# B&R Automation Studio project projekt_maszyny_grawerujacej
Automation Studio 4.7.2.98; technology packages: mapp 5.10.1, mappCockpit 5.10.1, mappMotion 5.10.1, mappView 5.10.1

## Configuration Config1

CPU X20CP0484, AutomationRuntime C4.72, Build 4.1.2, Safety 0.0, Vc V4.72.0

### Task classes (Cpu.sw)
```
Cyclic#2 (cycle 20000 us, tolerance 20000 us):
  Program1 <- Program1.prg
DataObjects: McAcpSys
NcDataObjects: IProg <- CNC.IProg.dob, isProg <- CNC.isProg.dob, WProg <- CNC.WProg.dob, UProg <- CNC.UProg.dob, XProg <- CNC.XProg.dob, RProg <- CNC.RProg.dob
Binaries: arcoal, arflatprv, arsvcreg, mvLoader, TCLang, TCData, McAcpSim, FWRules, McAcpDrv, udbdef, McMechSys, mCoWebSc, Config_3, arconfig, Settings, User, asfw, ashwd, Config_6, Config_1, ashwac, TC, Role, sysconf, Config_4, Config, Hierarchy, iomap, Config_2, Config_5
Libraries: McBase, MpCnc, MpBase, McAxGroup, McPathGen, McAxis, McProgInt, McAcpAx, MpAxis, CoTrace, AsZip, FileIO, runtime, MpAlarmX, astime, MpFile, MpServer, sys_lib, asarlog, asmem, asbrstr, asieccon, aruser, dataobj, powerlnk, asusb, brsystem, asarprof, arssl
```

### Hardware
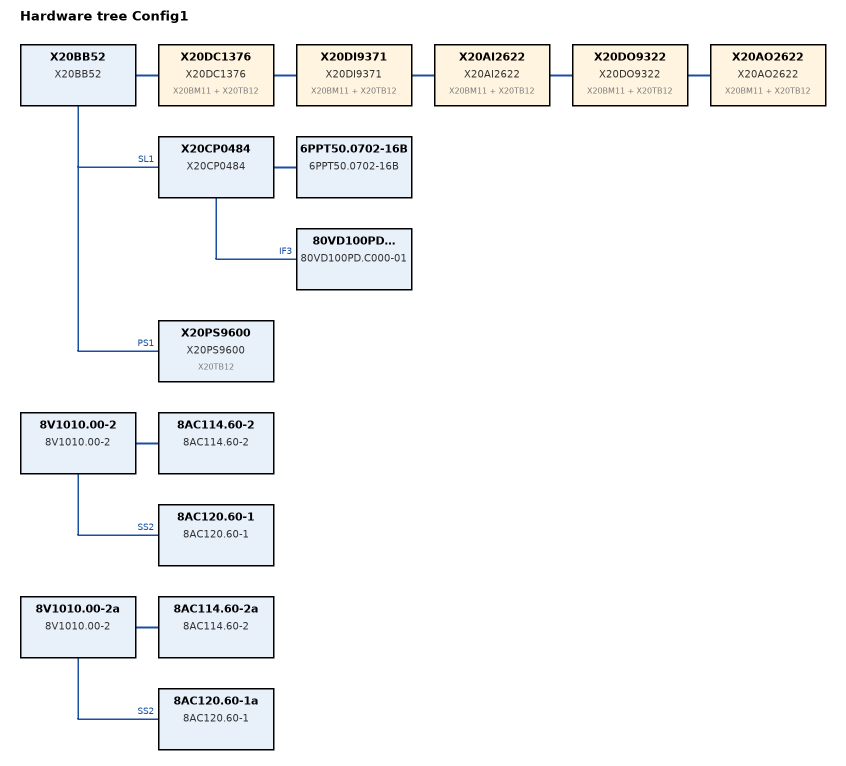
```
6PPT50.0702-16B : 6PPT50.0702-16B v1.0.0.0  [ETH1 -> X20CP0484.IF2 [Cable Type=PowerlinkCable, Length=10, Version=1.0.0.2]]
  Terminal = true
  PasswordVNC = 
  PasswordCIFS = 
  PasswordService = 
80VD100PD.C000-01 : 80VD100PD.C000-01 v2.4.0.0  [PLK1 -> X20CP0484.IF3 (NodeNumber=3) [Cable Type=PowerlinkCable, Length=10, Version=1.0.0.2]; PLK2 -> 8AC114.60-2a.PLK1 (NodeNumber=3) [Cable Type=PowerlinkCable, Length=10, Version=1.0.0.2]]
  DriveConfiguration/Module:
    McAcoposTypeID = AcoposMicroDConfig
    ActivateACOPOSSimulationOnPLC = 0
  DriveConfiguration/Channel[1]/RealAxis:
    AxisReference = gAxisQX
  DriveConfiguration/Channel[1]/RealAxis/MechanicalElements/Gearbox:
    InputIsReadOnly = 0
    Input = 1
    OutputIsReadOnly = 0
    Output = 1
  DriveConfiguration/Channel[1]/RealAxis/MechanicalElements/RotaryToLinearTransformation:
    ReferenceDistanceIsReadOnly = 0
    ReferenceDistance = 600
  DriveConfiguration/Channel[1]/RealAxis/Controller:
    ModeIsReadOnly = 0
    Mode = PositionController
  DriveConfiguration/Channel[1]/RealAxis/Controller/Mode/Position:
    ProportionalGain = 50.0
    IntegrationTime = 0.0
    PredictionTime = 0.0004
    TotalDelayTime = 0.0004
  DriveConfiguration/Channel[1]/RealAxis/Controller/Mode/Speed:
    ProportionalGainIsReadOnly = 0
    ProportionalGain = 2.0
    IntegrationTimeIsReadOnly = 0
    IntegrationTime = 0.0
    FilterTimeIsReadOnly = 0
    FilterTime = 0.0
  DriveConfiguration/Channel[1]/RealAxis/Controller/Mode/LoopFilters:
    LoopFilter1 = NotUsed
    LoopFilter2 = NotUsed
    LoopFilter3 = NotUsed
  DriveConfiguration/Channel[1]/RealAxis/Homing:
    Mode = Direct
  DriveConfiguration/Channel[1]/RealAxis/Homing/Mode:
    Position = 0.0
    ReferencePulse = NotUsed
  DriveConfiguration/Channel[1]/RealAxis/Homing:
    RestorePositionVariable = 
  DriveConfiguration/Channel[1]/RealAxis/StopReaction:
    Quickstop = DecelerationLimit
    DriveError = DecelerationLimit
  DriveConfiguration/Channel[1]/RealAxis/MovementErrorLimits:
    PositionError = 12.0
    VelocityErrorMonitoring = Automatic1
  DriveConfiguration/Channel[1]/RealAxis:
    JerkFilter = NotUsed
  DriveConfiguration/Channel[1]/RealAxis/DigitalInputs/HomingSwitch:
    Source = NotUsed
    Level = High
  DriveConfiguration/Channel[1]/RealAxis/DigitalInputs/PositiveLimitSwitch:
    Source = NotUsed
    Level = High
  DriveConfiguration/Channel[1]/RealAxis/DigitalInputs/NegativeLimitSwitch:
    Source = NotUsed
    Level = High
  DriveConfiguration/Channel[1]/RealAxis/DigitalInputs/Trigger1:
    Level = High
  DriveConfiguration/Channel[1]/RealAxis/DigitalInputs/Trigger2:
    Level = High
  DriveConfiguration/Channel[1]/RealAxis/DigitalInputs/Quickstop:
    Input = Trigger2
  DriveConfiguration/Channel[1]/RealAxis/Simulation:
    SimulationModeOnPLC = SetValueGeneration
    SimulationModeOnACOPOS = NotUsed
  DriveConfiguration/Channel[2]/RealAxis:
    AxisReference = gAxisQY
  DriveConfiguration/Channel[2]/RealAxis/MechanicalElements/Gearbox:
    InputIsReadOnly = 0
    Input = 1
    OutputIsReadOnly = 0
    Output = 1
  DriveConfiguration/Channel[2]/RealAxis/MechanicalElements/RotaryToLinearTransformation:
    ReferenceDistanceIsReadOnly = 0
    ReferenceDistance = 50
  DriveConfiguration/Channel[2]/RealAxis/Controller:
    ModeIsReadOnly = 0
    Mode = PositionController
  DriveConfiguration/Channel[2]/RealAxis/Controller/Mode/Position:
    ProportionalGain = 50.0
    IntegrationTime = 0.0
    PredictionTime = 0.0004
    TotalDelayTime = 0.0004
  DriveConfiguration/Channel[2]/RealAxis/Controller/Mode/Speed:
    ProportionalGainIsReadOnly = 0
    ProportionalGain = 2.0
    IntegrationTimeIsReadOnly = 0
    IntegrationTime = 0.0
    FilterTimeIsReadOnly = 0
    FilterTime = 0.0
  DriveConfiguration/Channel[2]/RealAxis/Controller/Mode/LoopFilters:
    LoopFilter1 = NotUsed
    LoopFilter2 = NotUsed
    LoopFilter3 = NotUsed
  DriveConfiguration/Channel[2]/RealAxis/Homing:
    Mode = Direct
  DriveConfiguration/Channel[2]/RealAxis/Homing/Mode:
    Position = 0.0
    ReferencePulse = NotUsed
  DriveConfiguration/Channel[2]/RealAxis/Homing:
    RestorePositionVariable = 
  DriveConfiguration/Channel[2]/RealAxis/StopReaction:
    Quickstop = DecelerationLimit
    DriveError = DecelerationLimit
  DriveConfiguration/Channel[2]/RealAxis/MovementErrorLimits:
    PositionError = 12.0
    VelocityErrorMonitoring = Automatic1
  DriveConfiguration/Channel[2]/RealAxis:
    JerkFilter = NotUsed
  DriveConfiguration/Channel[2]/RealAxis/DigitalInputs/HomingSwitch:
    Source = NotUsed
    Level = High
  DriveConfiguration/Channel[2]/RealAxis/DigitalInputs/PositiveLimitSwitch:
    Source = NotUsed
    Level = High
  DriveConfiguration/Channel[2]/RealAxis/DigitalInputs/NegativeLimitSwitch:
    Source = NotUsed
    Level = High
  DriveConfiguration/Channel[2]/RealAxis/DigitalInputs/Trigger1:
    Level = High
  DriveConfiguration/Channel[2]/RealAxis/DigitalInputs/Trigger2:
    Level = High
  DriveConfiguration/Channel[2]/RealAxis/DigitalInputs/Quickstop:
    Input = Trigger2
  DriveConfiguration/Channel[2]/RealAxis/Simulation:
    SimulationModeOnPLC = SetValueGeneration
    SimulationModeOnACOPOS = NotUsed
8AC114.60-2 : 8AC114.60-2 v1.0.0.8  [SS -> 8V1010.00-2.SS1; PLK1 -> 8AC114.60-2a.PLK2 [Cable Type=PowerlinkCable, Length=10, Version=1.0.0.2]]
8AC114.60-2a : 8AC114.60-2 v1.0.0.8  [SS -> 8V1010.00-2a.SS1; PLK1 -> 80VD100PD.C000-01.PLK2 [Cable Type=PowerlinkCable, Length=10, Version=1.0.0.2]; PLK2 -> 8AC114.60-2.PLK1 [Cable Type=PowerlinkCable, Length=10, Version=1.0.0.2]]
8AC120.60-1 : 8AC120.60-1 v2.2.0.0  [SS -> 8V1010.00-2.SS2]
  PlugInType = Encoder
  McAcoposTypeID = AcoposPlugInConfig
8AC120.60-1a : 8AC120.60-1 v2.2.0.0  [SS -> 8V1010.00-2a.SS2]
  PlugInType = Encoder
  McAcoposTypeID = AcoposPlugInConfig
8V1010.00-2 : 8V1010.00-2 v2.2.0.0
  DriveConfiguration/Module:
    McAcoposTypeID = AcoposConfig
    ActivateACOPOSSimulationOnPLC = 0
  DriveConfiguration/Channel[1]/RealAxis:
    AxisReference = gAxisQS
  DriveConfiguration/Channel[1]/RealAxis/MechanicalElements/Gearbox:
    InputIsReadOnly = 0
    Input = 1
    OutputIsReadOnly = 0
    Output = 1
  DriveConfiguration/Channel[1]/RealAxis/MechanicalElements/RotaryToLinearTransformation:
    ReferenceDistanceIsReadOnly = 0
    ReferenceDistance = 600
  DriveConfiguration/Channel[1]/RealAxis/Controller:
    ModeIsReadOnly = 0
    Mode = PositionController
  DriveConfiguration/Channel[1]/RealAxis/Controller/Mode/Position:
    ProportionalGain = 50.0
    IntegrationTime = 0.0
    PredictionTime = 0.0004
    TotalDelayTime = 0.0004
  DriveConfiguration/Channel[1]/RealAxis/Controller/Mode/Speed:
    ProportionalGainIsReadOnly = 0
    ProportionalGain = 2.0
    IntegrationTimeIsReadOnly = 0
    IntegrationTime = 0.0
    FilterTimeIsReadOnly = 0
    FilterTime = 0.0
  DriveConfiguration/Channel[1]/RealAxis/Controller/Mode/LoopFilters:
    LoopFilter1 = NotUsed
    LoopFilter2 = NotUsed
    LoopFilter3 = NotUsed
  DriveConfiguration/Channel[1]/RealAxis/Homing:
    Mode = Direct
  DriveConfiguration/Channel[1]/RealAxis/Homing/Mode:
    Position = 0.0
    ReferencePulse = NotUsed
  DriveConfiguration/Channel[1]/RealAxis/Homing:
    RestorePositionVariable = 
  DriveConfiguration/Channel[1]/RealAxis/StopReaction:
    Quickstop = DecelerationLimit
    DriveError = DecelerationLimit
  DriveConfiguration/Channel[1]/RealAxis/MovementErrorLimits:
    PositionError = 12.0
    VelocityErrorMonitoring = Automatic1
  DriveConfiguration/Channel[1]/RealAxis:
    JerkFilter = NotUsed
  DriveConfiguration/Channel[1]/RealAxis/DigitalInputs/HomingSwitch:
    Level = High
  DriveConfiguration/Channel[1]/RealAxis/DigitalInputs/PositiveLimitSwitch:
    Level = High
  DriveConfiguration/Channel[1]/RealAxis/DigitalInputs/NegativeLimitSwitch:
    Level = High
  DriveConfiguration/Channel[1]/RealAxis/DigitalInputs/Trigger1:
    Level = High
  DriveConfiguration/Channel[1]/RealAxis/DigitalInputs/Trigger2:
    Level = High
  DriveConfiguration/Channel[1]/RealAxis/DigitalInputs/Quickstop:
    Input = Trigger2
  DriveConfiguration/Channel[1]/RealAxis/Simulation:
    SimulationModeOnPLC = SetValueGeneration
    SimulationModeOnACOPOS = NotUsed
8V1010.00-2a : 8V1010.00-2 v2.2.0.0
  DriveConfiguration/Module:
    McAcoposTypeID = AcoposConfig
    ActivateACOPOSSimulationOnPLC = 0
  DriveConfiguration/Channel[1]/RealAxis:
    AxisReference = gAxisQZ
  DriveConfiguration/Channel[1]/RealAxis/MechanicalElements/Gearbox:
    InputIsReadOnly = 0
    Input = 1
    OutputIsReadOnly = 0
    Output = 1
  DriveConfiguration/Channel[1]/RealAxis/MechanicalElements/RotaryToLinearTransformation:
    ReferenceDistanceIsReadOnly = 0
    ReferenceDistance = 50
  DriveConfiguration/Channel[1]/RealAxis/Controller:
    ModeIsReadOnly = 0
    Mode = PositionController
  DriveConfiguration/Channel[1]/RealAxis/Controller/Mode/Position:
    ProportionalGain = 50.0
    IntegrationTime = 0.0
    PredictionTime = 0.0004
    TotalDelayTime = 0.0004
  DriveConfiguration/Channel[1]/RealAxis/Controller/Mode/Speed:
    ProportionalGainIsReadOnly = 0
    ProportionalGain = 2.0
    IntegrationTimeIsReadOnly = 0
    IntegrationTime = 0.0
    FilterTimeIsReadOnly = 0
    FilterTime = 0.0
  DriveConfiguration/Channel[1]/RealAxis/Controller/Mode/LoopFilters:
    LoopFilter1 = NotUsed
    LoopFilter2 = NotUsed
    LoopFilter3 = NotUsed
  DriveConfiguration/Channel[1]/RealAxis/Homing:
    Mode = Direct
  DriveConfiguration/Channel[1]/RealAxis/Homing/Mode:
    Position = 300.0
    ReferencePulse = NotUsed
  DriveConfiguration/Channel[1]/RealAxis/Homing:
    RestorePositionVariable = 
  DriveConfiguration/Channel[1]/RealAxis/StopReaction:
    Quickstop = DecelerationLimit
    DriveError = DecelerationLimit
  DriveConfiguration/Channel[1]/RealAxis/MovementErrorLimits:
    PositionError = 12.0
    VelocityErrorMonitoring = Automatic1
  DriveConfiguration/Channel[1]/RealAxis:
    JerkFilter = NotUsed
  DriveConfiguration/Channel[1]/RealAxis/DigitalInputs/HomingSwitch:
    Level = High
  DriveConfiguration/Channel[1]/RealAxis/DigitalInputs/PositiveLimitSwitch:
    Level = High
  DriveConfiguration/Channel[1]/RealAxis/DigitalInputs/NegativeLimitSwitch:
    Level = High
  DriveConfiguration/Channel[1]/RealAxis/DigitalInputs/Trigger1:
    Level = High
  DriveConfiguration/Channel[1]/RealAxis/DigitalInputs/Trigger2:
    Level = High
  DriveConfiguration/Channel[1]/RealAxis/DigitalInputs/Quickstop:
    Input = Trigger2
  DriveConfiguration/Channel[1]/RealAxis/Simulation:
    SimulationModeOnPLC = SetValueGeneration
    SimulationModeOnACOPOS = NotUsed
X20AI2622 : X20AI2622 v1.0.4.0  [SS1 -> X20TB12d.SS; SL -> X20BM11c.SL1]
X20AO2622 : X20AO2622 v1.1.0.0  [SS1 -> X20TB12e.SS; SL -> X20BM11d.SL1]
X20BB52 : X20BB52 v1.1.0.0
X20BM11 : X20BM11 v1.0.0.1  [X2X1 -> X20BM11b.X2X2]
X20BM11a : X20BM11 v1.0.0.1  [X2X1 -> X20BM11c.X2X2]
X20BM11b : X20BM11 v1.0.0.1  [X2X1 -> X20BB52.IF6]
X20BM11c : X20BM11 v1.0.0.1  [X2X1 -> X20BM11.X2X2]
X20BM11d : X20BM11 v1.0.0.1  [X2X1 -> X20BM11a.X2X2]
X20CP0484 : X20CP0484 v1.2.1.0  [SL -> X20BB52.SL1]
  Connector IF2:
    ActivateDevice = 1
  Connector IF3:
    InternetAddress = 10.0.0.10
  ConfigurationID = projekt_maszyny_grawerującej_Config1
  UserPartitionSize = 2
  AutomaticTransferOfUserfiles = on
  Simulation = 1
  TimerDeviceType = EPLX2X
  TimerDevice = X20CP0484.IF3
  TaskClassIdleTime = 2000
  Cyclic1Duration = 2000
  Cyclic1Tolerance = 0
  Cyclic1Stack = 32000
  Cyclic2Duration = 20000
  Cyclic2Tolerance = 20000
  Cyclic3Duration = 50000
  Cyclic3Tolerance = 50000
  Cyclic4Duration = 100000
  Cyclic4Tolerance = 100000
  Cyclic5Duration = 200000
  Cyclic5Tolerance = 200000
  Cyclic6Duration = 500000
  Cyclic6Tolerance = 500000
  Cyclic7Duration = 1000000
  Cyclic7Tolerance = 1000000
  Cyclic8Duration = 10000
  Cyclic8Tolerance = 30000000
  ActivateSntpServer = 1
  ActivateSntp = 1
  SntpcServAddr2 = 10.0.0,5
  ActivateOpcUa = 1
  OpcUaInformationModels_PV_Version = 1
X20DC1376 : X20DC1376 v1.0.2.0  [SS1 -> X20TB12c.SS; SL -> X20BM11b.SL1]
X20DI9371 : X20DI9371 v1.0.2.0  [SS1 -> X20TB12a.SS; SL -> X20BM11.SL1]
X20DO9322 : X20DO9322 v1.1.0.0  [SS1 -> X20TB12b.SS; SL -> X20BM11a.SL1]
X20PS9600 : X20PS9600 v1.0.1.0  [PS -> X20BB52.PS1; SS1 -> X20TB12.SS]
X20TB12 : X20TB12 v1.0.0.0
X20TB12a : X20TB12 v1.0.0.0
X20TB12b : X20TB12 v1.0.0.0
X20TB12c : X20TB12 v1.0.0.0
X20TB12d : X20TB12 v1.0.0.0
X20TB12e : X20TB12 v1.0.0.0
```

### IoMap.iom - X20CP0484/IoMap.iom
```iecst
VAR_CONFIG
	::gdoProcessLamp AT %QX."X20DO9322".DigitalOutput01;
	::gdoMillingLamp AT %QX."X20DO9322".DigitalOutput02;
	::Program1:Sensor AT %IX."X20DI9371".DigitalInput01;
END_VAR
```

### Config_1.axesgroup - X20CP0484/mappMotion/3AxesCNCXYZ/Config_1.axesgroup
```
Element gCncXYZ (Type=axesgroup)
  Type = PathGenAxesGroup
    ProcessingTaskClass = 1
    License = 1
    PhysicalAxes:
      JointAxes:
        JointAxis[1]:
          Name = QX
          AxisRef = gAxisQX
        JointAxis[2]:
          Name = QY
          AxisRef = gAxisQY
        JointAxis[3]:
          Name = QZ
          AxisRef = gAxisQZ
      SlaveAxes:
        SlaveAxis[1]:
          Name = QS
          AxisRef = gAxisQS
    MechanicalSystem:
      MechSysRef = MechSys_3AxCNCXYZ
    BasicSettings:
      ModalDataBehaviour = ResetToDefault
      GeometryPlanning:
        RoundingMode = Standard
        MaxCornerDeviation = 0.0
        MaxTangentialTransitionDeviation = 0.0
        MaxRadiusDeviation = 0.001
        WorkingPlane = XY
      TrajectoryPlanning = Basic
        LimitCheckResolution = UserDefinedTime
          Time = 0.01
        BufferTime = UserDefinedTime
          Time = 0.1
    AxesGroupFeatures:
      FeatureRef[1] = Feature_Programs
      FeatureRef[2] = Feature_Jogging
      FeatureRef[3] = Feature_spindles
  Alarms = None
```

### Config_2.axis - X20CP0484/mappMotion/3AxesCNCXYZ/Config_2.axis
```
Element gAxisQX (Type=axis)
  BaseTypeIsReadOnly = 0
  BaseType = Linear
    MeasurementUnit = 5066068
    MeasurementResolutionIsReadOnly = 0
    MeasurementResolution = 0.01
    CountDirectionIsReadOnly = 0
    CountDirection = Standard
  MovementLimitsIsReadOnly = 0
  MovementLimits = Internal
    Position:
      LowerLimitMin = -1.79769313486231E308
      UpperLimitMax = 1.79769313486231E308
      LowerLimit = -1000.0
      UpperLimit = 1000.0
    VelocityIsReadOnly = 0
    Velocity:
      VelocityMax = 3.4E38
      Velocity = 10000.0
    AccelerationIsReadOnly = 0
    Acceleration:
      AccelerationMax = 3.4E38
      Acceleration = 100000.0
    DecelerationIsReadOnly = 0
    Deceleration:
      DecelerationMax = 3.4E38
      Deceleration = 100000.0
  Alarms = MpAlarmX
Element gAxisQY (Type=axis)
  BaseTypeIsReadOnly = 0
  BaseType = LinearBounded
    MeasurementUnit = 5066068
    MeasurementResolutionIsReadOnly = 0
    MeasurementResolution = 0.01
    CountDirectionIsReadOnly = 0
    CountDirection = Standard
  MovementLimitsIsReadOnly = 0
  MovementLimits = Internal
    Position:
      LowerLimitMin = -1.79769313486231E308
      UpperLimitMax = 1.79769313486231E308
      LowerLimit = -100.0
      UpperLimit = 400.0
    VelocityIsReadOnly = 0
    Velocity:
      VelocityMax = 3.4E38
      Velocity = 10000.0
    AccelerationIsReadOnly = 0
    Acceleration:
      AccelerationMax = 3.4E38
      Acceleration = 100000.0
    DecelerationIsReadOnly = 0
    Deceleration:
      DecelerationMax = 3.4E38
      Deceleration = 100000.0
  Alarms = MpAlarmX
Element gAxisQZ (Type=axis)
  BaseTypeIsReadOnly = 0
  BaseType = LinearBounded
    MeasurementUnit = 5066068
    MeasurementResolutionIsReadOnly = 0
    MeasurementResolution = 0.01
    CountDirectionIsReadOnly = 0
    CountDirection = Standard
  MovementLimitsIsReadOnly = 0
  MovementLimits = Internal
    Position:
      LowerLimitMin = -1.79769313486231E308
      UpperLimitMax = 1.79769313486231E308
      LowerLimit = 0
      UpperLimit = 300
    VelocityIsReadOnly = 0
    Velocity:
      VelocityMax = 3.4E38
      Velocity = 10000.0
    AccelerationIsReadOnly = 0
    Acceleration:
      AccelerationMax = 3.4E38
      Acceleration = 100000.0
    DecelerationIsReadOnly = 0
    Deceleration:
      DecelerationMax = 3.4E38
      Deceleration = 100000.0
  Alarms = MpAlarmX
Element gAxisQS (Type=axis)
  BaseTypeIsReadOnly = 0
  BaseType = Rotary
    MeasurementUnitIsReadOnly = 0
    MeasurementUnit = 5059636
    MeasurementResolutionIsReadOnly = 0
    MeasurementResolution = 0.01
    CountDirectionIsReadOnly = 0
    CountDirection = Standard
  MovementLimitsIsReadOnly = 0
  MovementLimits = Internal
    Position:
      LowerLimitMin = -1.79769313486231E308
      UpperLimitMax = 1.79769313486231E308
      LowerLimit = -1000.0
      UpperLimit = 1000.0
    VelocityIsReadOnly = 0
    Velocity:
      VelocityMax = 3.4E38
      Velocity = 250.0
    AccelerationIsReadOnly = 0
    Acceleration:
      AccelerationMax = 3.4E38
      Acceleration = 500.0
    DecelerationIsReadOnly = 0
    Deceleration:
      DecelerationMax = 3.4E38
      Deceleration = 500.0
  Alarms = MpAlarmX
```

### Config_3.mechanicalsystem - X20CP0484/mappMotion/3AxesCNCXYZ/Config_3.mechanicalsystem
```
Element MechSys_3AxCNCXYZ (Type=mechanicalsystem)
  Type = 3AxesCNC
    Subtype = 3AxesCNCXYZ
      CoordinatesNames = Default
        XCoordinateName = X
        YCoordinateName = Y
        ZCoordinateName = Z
      WireFrameModel = Standard
        FlangeToTcp = ConnectionLine
          Distance = 0.0
      JointAxesPositionLimits:
        JointAxis[1] = UseAxisLimits
        JointAxis[2] = UseAxisLimits
        JointAxis[3] = UseAxisLimits
```

### Config_4.axesgroupfeature - X20CP0484/mappMotion/3AxesCNCXYZ/Config_4.axesgroupfeature
```
Element Feature_Programs (Type=axesgroupfeature)
  Type = Program
    ModalDataBehaviour = UseAxesGroupSettings
    InitialSettings:
      InterpolationTypes = LinearRapid
      PositionCoordinates = Absolute
      CircleCoordinates = Relative
      JACS_ACSProgramming = JACS
      ContourConnection = Inactive
      ProgrammingUnits = UseAxesGroupSettings
      Feedrates:
        FeedCharacteristic = StandardCharacteristic
        FeedType = Feedrate
        FeedReduction = Inactive
        FeedrateValue = 0.0
        InverseFeedrateValue = 0.0
        FeedratePerRevValue = 0.0
    DefaultLanguage = BRGCode
    Location = Default
      FileDevice = CNC_PrgDir
Element Feature_Jogging (Type=axesgroupfeature)
  Type = Jogging
Element Feature_spindles (Type=axesgroupfeature)
  Type = Spindles
    ModalDataBehaviour = UseAxesGroupSettings
    Spindle[1]:
      SlaveAxisName = QS
```

### Config.mpalarmxcore - X20CP0484/mappServices/Config.mpalarmxcore
```
Element gAlarmXCore (Type=mpalarmxcore)
  mapp.AlarmX.Core.Configuration:
    [0]:
      Name = EmergButton
      Message = Emergency button has been pushed
      Severity = 20
    [1]:
      Name = Elem2Small
      Message = Element is too small
      Severity = 10
    [2]:
      Name = PowerOff
      Message = Unexpected  Power Off  event
      Severity = 20
```

## Logical view

Binary libraries used (declarations not repeated): operator, runtime, astime, AsIecCon, McBase, MpCnc 5.10.1, MpBase, McAxGroup 5.10.1, McPathGen 5.10.1, McAxis, McProgInt 5.10.1, McAcpAx, MpAxis, CoTrace 5.10.0, AsZip, FileIO, MpAlarmX 5.10.1, MpFile 5.10.1, MpServer 5.10.0

### Global.typ - Global data types
```iecst
TYPE
	InType : 	STRUCT
		gdiStopButton : BOOL; (*emergency mechine stopping (INPUT)*)
		gdiObjSensor : BOOL; (*the vaule is TRUE if sensor detects object (INPUT)*)
	END_STRUCT;
	OutType : 	STRUCT
		gdoMillingLamp : BOOL; (*Lamp is on ig milling cutter is revolving (OUTPUT)*)
		gdoProcessLamp : BOOL; (*Lamp is ON if obj is being processed (OUTPUT)*)
	END_STRUCT;
END_TYPE
```

### Global.var - Global variables
```iecst
VAR
	gdiStopButton : BOOL; (*emergency mechine stopping (INPUT)*)
	gdiObjSensor : BOOL; (*the vaule is TRUE if sensor detects object (INPUT)*)
	gdoMillingLamp : BOOL; (*Lamp is on ig milling cutter is revolving (OUTPUT)*)
	gdoProcessLamp : BOOL; (*Lamp is ON if obj is being processed (OUTPUT)*)
END_VAR
```


### Program Logical/Program1 (IEC)

#### Types.typ
```iecst
TYPE
	JogStatusEnum :
		(
		JOGTYPE,
		XUP,
		XDOWN,
		YUP,
		YDOWN,
		ZUP,
		ZDOWN
		);
	WorkingModeEnum :
		(
		CHOOSE_MODE,
		AUTOMATIC,
		MANUAL,
		STOP
		);
	ServoStatusEnum :
		(
		POWER_OFF := 0,
		POWER_ON := 1,
		HOME := 2,
		READY_TO_WORK := 3
		);
	AutoModeStatusEnum :
		(
		XMOVING,
		WORKING,
		ASIGNSTART,
		CALCSIZE,
		ASIGNEND
		);
	ChooseProgrEnum :
		(
		CAPITAL_I := 0,
		SMALL_I := 1,
		CAPITAL_W := 2,
		CAPITAL_U := 3,
		CAPITAL_X := 4,
		CAPITAL_R := 5
		);
	ManualModeStatusEnum :
		(
		JOG,
		PRECISE
		);
	AsignPropEnum :
		(
		AXIS2MOVE,
		MOVEX,
		MOVEY,
		MOVEZ,
		MOVES
		);
END_TYPE
```

#### Variables.var
```iecst
(*axis and program configuration and functionality*)
VAR
	MpCnc3Axis_0 : MpCnc3Axis; (*3 axis Group*)
	Xaxis : MpAxisBasic; (*X axis func*)
	Yaxis : MpAxisBasic; (*Y axis func*)
	Zaxis : MpAxisBasic; (*Z axis func*)
	Saxis : MpAxisBasic; (*S axis func*)
	CncParameters_3Axis : MpCnc3AxisParType; (*axis group parameters*)
	X_param : MpAxisBasicParType; (*X axis parameters*)
	Y_param : MpAxisBasicParType; (*Y axis parameters*)
	Z_param : MpAxisBasicParType; (*Z axis parameters*)
	S_param : MpAxisBasicParType; (*S axis parameters*)
	ServoStatus : ServoStatusEnum; (*machine states*)
	WorkingMode : WorkingModeEnum; (*woking mode states*)
END_VAR
(*automatic mode*)
VAR
	AutoModeStatus : AutoModeStatusEnum; (*automatic mode states*)
	ChooseProgr : ChooseProgrEnum; (*enum with cnc programs*)
	StopMode : BOOL; (*ON/OFF stop mode*)
	AutomaticON : BOOL; (*ON/OFF automatic mode*)
	Sensor : BOOL; (*Sensor on off*)
	LengthStart : LREAL; (*start obj position*)
	LengthEnd : LREAL; (*end obj position*)
	ChooseElemNumber : USINT;
	Elements2Done : INT; (*processed elements*)
	NumOfElem : INT; (*Choose number of elem to process*)
	ObjLength : LREAL; (*length of obj*)
	CentreX : LREAL; (*obj centre X axis*)
END_VAR
VAR CONSTANT
	CentreY : LREAL := 200; (*obj centre Y axis*)
END_VAR
(*manual mode*)
VAR
	ManualON : BOOL; (*ON/oFF Manual mode*)
	ManualModeStatus : ManualModeStatusEnum; (*manual mode states*)
	ManXPos : LREAL; (*choose x pos*)
	ManYPos : LREAL; (*choose y pos*)
	ManZPos : LREAL; (*choose z pos*)
	ManSPos : LREAL; (*choose s pos*)
	ManXVel : REAL; (*choose x vel*)
	AsignProp : AsignPropEnum; (*states in which y can choose axis to move in manual mode*)
	ManYVel : REAL; (*choose y vel*)
	ManZVel : REAL; (*choose z vel*)
	ManSVel : REAL; (*choose s vel*)
	X2Move : BOOL; (*choose x axis to move*)
	Y2Move : BOOL; (*choose y axis to move*)
	Z2Move : BOOL; (*choose z axis to move*)
	S2Move : BOOL; (*choose s axis to move*)
	Moveaxis : BOOL; (*comfirms axis move in manual mode*)
END_VAR
(*jogging*)
VAR
	JogStatus : JogStatusEnum; (*jog mode states*)
	JogUpX : BOOL; (*jog x forward*)
	JogDownX : BOOL; (*jog x backward*)
	JogUpY : BOOL; (*jog y forward*)
	JogDownY : BOOL; (*jog y backward*)
	JogUpZ : BOOL; (*jog z gorward*)
	JogDownZ : BOOL; (*jog z backward*)
	JogUpS : BOOL; (*jog s forward*)
	JogDownS : BOOL; (*jog s backward*)
	JogModeOn : BOOL; (*on offf joging mode*)
END_VAR
(*visualization (variables needed to show process icons)*)
VAR
	Proccessing : BOOL;
	YOff : BOOL;
	Ymove : BOOL;
	YOn : BOOL;
	XOff : BOOL;
	Xmove : BOOL;
	XOn : BOOL;
	ZOff : BOOL;
	Zmove : BOOL;
	ZOn : BOOL;
	SOff : BOOL;
	Smove : BOOL;
	SOn : BOOL;
	ActMode4MV : STRING[80]; (*Helps display actual mode in mappView *)
END_VAR
(*AlarmSystem*)
VAR
	EmergStop : BOOL; (*Emergency Stop Button. Stops machine *)
	MpAlarmXCore_0 : MpAlarmXCore;
END_VAR
VAR CONSTANT
	cmdErrorReset : BOOL := FALSE;
END_VAR
VAR
	SetAlarmEmerg : USINT;
	cmdSetAlarm : BOOL;
	AckALL : MpAlarmXAcknowledgeAll;
	EmergStopAck : BOOL;
	AckAllButton : BOOL;
	Elem2SmallAck : BOOL;
	Elem2Small : BOOL;
	WarningSymbol1 : BOOL;
	WarningSymbol2 : BOOL;
	ShowWarning : BOOL;
END_VAR
(*Alarm History*)
VAR
	MpAlarmXHistory_0 : MpAlarmXHistory;
	MpAlarmXHistoryUI_0 : MpAlarmXHistoryUI;
	MpAlarmXListUI_0 : MpAlarmXListUI;
	MpAlarmXListUIConnectType_0 : MpAlarmXListUIConnectType;
	AlarmXHistoryUIConnect : MpAlarmXHistoryUIConnectType;
END_VAR
(*Visualization plc Open state*)
VAR
	XState : STRING[80];
	YState : STRING[80];
	ZState : STRING[80];
	SState : STRING[80];
END_VAR
```

#### Main.st
```iecst
(*************************************************************
* COPYRIGHT – B&R Industrial Automation
 *************************************************************
* PROGRAM: Milling Machine
* Author: Patrtyk Tomaszewski
* Created: 10/8/2020
*************************************************************
* Project Milling Machine
*************************************************************)

PROGRAM _INIT
	//Alarms
	MpAlarmXCore_0.MpLink := ADR(gAlarmXCore);
	MpAlarmXCore_0.Enable := TRUE;
	AckALL.MpLink := ADR(gAlarmXCore);
	AckALL.Enable := TRUE;
	//Alarm History

	MpAlarmXHistory_0.MpLink := ADR(gAlarmXHistory);
	MpAlarmXHistory_0.Enable := TRUE;
	MpAlarmXHistory_0.DeviceName := ADR('CF');

	//3 axis
	MpCnc3Axis_0.MpLink := ADR(gCncXYZ);
	MpCnc3Axis_0.Enable := TRUE;
	MpCnc3Axis_0.Parameters := ADR(CncParameters_3Axis);
	MpCnc3Axis_0.Override := 100.0;
	///////////////////////////////

	//X axis
	Xaxis.MpLink := ADR(gAxisQX);
	Xaxis.Parameters := ADR(X_param);
	Xaxis.Enable := TRUE;
	X_param.Velocity := 30.0;
	X_param.Acceleration := 50.0;
	X_param.Deceleration := 50.0;
	X_param.Homing.Mode := mcHOMING_DEFAULT;
   /////

	//Y axis
	Yaxis.MpLink := ADR(gAxisQY);
	Yaxis.Parameters := ADR(Y_param);
	Yaxis.Enable := TRUE;
	Y_param.Velocity := 30.0;
	Y_param.Acceleration := 50.0;
	Y_param.Deceleration := 50.0;
	Y_param.Homing.Mode := mcHOMING_DEFAULT;
	/////

	//Z axis
	Zaxis.MpLink := ADR(gAxisQZ);
	Zaxis.Parameters := ADR(Z_param);
	Zaxis.Enable := TRUE;
	Z_param.Velocity := 30.0;
	Z_param.Acceleration := 50.0;
	Z_param.Deceleration := 50.0;
	Z_param.Homing.Mode := mcHOMING_DEFAULT;
	/////

	//S axis
	Saxis.MpLink := ADR(gAxisQS);
	Saxis.Parameters := ADR(S_param);
	Saxis.Enable := TRUE;
	S_param.Velocity := 166.6;
	S_param.Acceleration := 400.0;
	S_param.Deceleration := 400.0;
	S_param.Homing.Mode := mcHOMING_DEFAULT;
	S_param.Jog.Velocity := 166.6;
	S_param.Jog.Acceleration := 400.0;
	S_param.Jog.Deceleration := 400.0;

	/////

END_PROGRAM

PROGRAM _CYCLIC

	(*
	Powering On Servo*)

	CASE ServoStatus OF

		POWER_OFF:
			ActMode4MV := 'POWER OFF';
			MpCnc3Axis_0.Update := TRUE;
			Xaxis.Power := FALSE;
			Yaxis.Power := FALSE;
			Zaxis.Power := FALSE;
			Saxis.Power := FALSE;
			StopMode := FALSE;
			ManualON := FALSE;
			AutomaticON := FALSE;
			IF  MpCnc3Axis_0.Info.ReadyToPowerOn AND MpCnc3Axis_0.Power THEN
				MpCnc3Axis_0.Update := FALSE;
				ServoStatus := POWER_ON;

			END_IF

		POWER_ON:
			ActMode4MV := 'POWER ON';
			MpCnc3Axis_0.Update := TRUE;
			Xaxis.Power := TRUE;
			Yaxis.Power := TRUE;
			Zaxis.Power := TRUE;
			Saxis.Power := TRUE;
			IF  MpCnc3Axis_0.PowerOn AND Xaxis.PowerOn AND Yaxis.PowerOn AND Zaxis.PowerOn AND Saxis.PowerOn THEN;
				MpCnc3Axis_0.Update := FALSE;
				ServoStatus := HOME;

			END_IF

		HOME:
			ActMode4MV := 'Homing';
			MpCnc3Axis_0.Home := TRUE;
			IF  MpCnc3Axis_0.IsHomed AND Xaxis.Position = 0.0 AND Yaxis.Position = 0.0 AND Zaxis.Position = 300.0 THEN;
				ActMode4MV := 'Ready To Work';
				ServoStatus := READY_TO_WORK;

			END_IF
		READY_TO_WORK:
			MpCnc3Axis_0.Home := FALSE;

			CASE WorkingMode OF

				CHOOSE_MODE:
					IF AutomaticON THEN;
						WorkingMode := AUTOMATIC;
						Elements2Done := 0;
					ELSIF ManualON THEN;
						WorkingMode := MANUAL;
					END_IF

				AUTOMATIC:
					AutomaticON := TRUE;
					MpCnc3Axis_0.Power := TRUE;
					ManualON := FALSE;

					ActMode4MV := 'Automatic Mode';
					CASE AutoModeStatus OF
						////////Const X axis move until we find elem
						XMOVING:
							Elem2Small := FALSE;
							X_param.Velocity := 30.0;
							Xaxis.Update := TRUE;
							IF Sensor = FALSE THEN;
								Xaxis.Update := FALSE;
								Xaxis.MoveVelocity := TRUE;
								IF StopMode THEN
									Xaxis.MoveVelocity := FALSE;
									AutomaticON := FALSE;
									NumOfElem := 0;
									WorkingMode := STOP;

								END_IF;

							ELSE
								gdoProcessLamp := TRUE;
								AutoModeStatus := ASIGNSTART;
							END_IF
							///////////////////////////

							///Calculate Length of element

						ASIGNSTART:
							X_param.Velocity := 20.0;
							Xaxis.Update := TRUE;
							LengthStart := Xaxis.Position;
							AutoModeStatus := ASIGNEND;

						ASIGNEND:
							Xaxis.Update := FALSE;
							IF Sensor = FALSE THEN;
								LengthEnd := Xaxis.Position;
								AutoModeStatus := CALCSIZE;
							END_IF

						CALCSIZE:
							ObjLength := LengthEnd - LengthStart;
							CentreX := LengthStart + (ObjLength / 2);
							AutoModeStatus := WORKING;
							/////////////////////////////////////

							///start program
						WORKING:
							Xaxis.MoveVelocity := FALSE;
							X_param.Velocity := 30.0;
							//Program I
							IF ChooseProgr = CAPITAL_I THEN

								IF ObjLength < 40 THEN
									Elem2Small := TRUE;
									gdoProcessLamp := FALSE;
									AutoModeStatus := XMOVING;

								ELSE
									X_param.Position := CentreX;
									Xaxis.Update := TRUE;
									Xaxis.MoveAbsolute := TRUE;

									IF  Xaxis.InPosition  THEN;
										Xaxis.Update := FALSE;
										Xaxis.MoveAbsolute := FALSE;
										CncParameters_3Axis.ProgramName := 'IProg';
										MpCnc3Axis_0.Update := TRUE;
										MpCnc3Axis_0.MoveProgram := TRUE;
										IF MpCnc3Axis_0.MoveDone THEN
											MpCnc3Axis_0.Update := FALSE;
											MpCnc3Axis_0.MoveProgram := FALSE;
											X_param.Position := LengthEnd;
											Xaxis.Update := TRUE;
											Xaxis.MoveAbsolute := TRUE;
											IF Xaxis.InPosition THEN
												Xaxis.Update := FALSE;
												Xaxis.MoveAbsolute := FALSE;
												IF StopMode THEN
													AutomaticON := FALSE;
													gdoProcessLamp := FALSE;
													NumOfElem := 0;
													WorkingMode := STOP;////////going to stop mode after completing program

												ELSE
													gdoProcessLamp := FALSE;
													Elements2Done := Elements2Done + 1;
													IF (Elements2Done = NumOfElem) AND (NumOfElem <> 0.0) THEN;
														NumOfElem := 0;
														Elements2Done := 0;
														StopMode := TRUE;
														AutomaticON := FALSE;
														WorkingMode := STOP;
													ELSE
														IF NumOfElem = 0.0 THEN;
															Elements2Done := FALSE;
															AutoModeStatus := XMOVING;
														ELSE
															AutoModeStatus := XMOVING;
														END_IF;
													END_IF;
												END_IF;

											END_IF;
										END_IF;
									END_IF;
								END_IF;
								//Program i
							ELSIF ChooseProgr = SMALL_I THEN

								IF ObjLength < 40 THEN
									Elem2Small := TRUE;
									gdoProcessLamp := FALSE;
									AutoModeStatus := XMOVING;
								ELSE

									X_param.Position := CentreX;
									Xaxis.Update := TRUE;
									Xaxis.MoveAbsolute := TRUE;
									IF Xaxis.InPosition THEN;
										Xaxis.Update := FALSE;
										Xaxis.MoveAbsolute := FALSE;
										CncParameters_3Axis.ProgramName := 'isProg';
										MpCnc3Axis_0.Update := TRUE;
										MpCnc3Axis_0.MoveProgram := TRUE;
										IF MpCnc3Axis_0.MoveDone THEN
											MpCnc3Axis_0.Update := FALSE;
											MpCnc3Axis_0.MoveProgram := FALSE;
											X_param.Position := LengthEnd;
											Xaxis.Update := TRUE;
											Xaxis.MoveAbsolute := TRUE;
											IF Xaxis.InPosition THEN
												Xaxis.Update := FALSE;
												Xaxis.MoveAbsolute := FALSE;
												IF StopMode THEN
													gdoProcessLamp := FALSE;
													AutomaticON := FALSE;
													NumOfElem := 0;
													WorkingMode := STOP;////////going to stop mode after completing program
												ELSE
													gdoProcessLamp := FALSE;
													Elements2Done := Elements2Done + 1;
													IF (Elements2Done = NumOfElem) AND (NumOfElem <> 0.0) THEN;
														NumOfElem := 0;
														Elements2Done := 0;
														StopMode := TRUE;
														AutomaticON := FALSE;
														WorkingMode := STOP;
													ELSE
														IF NumOfElem = 0.0 THEN;
															Elements2Done := FALSE;
															AutoModeStatus := XMOVING;
														ELSE
															AutoModeStatus := XMOVING;
														END_IF;
													END_IF;
												END_IF;

											END_IF;
										END_IF;
									END_IF;
								END_IF;
								///Program W
							ELSIF ChooseProgr = CAPITAL_W THEN
								IF ObjLength < 140 THEN
									Elem2Small := TRUE;
									gdoProcessLamp := FALSE;
									AutoModeStatus := XMOVING;
								ELSE

									X_param.Position := CentreX + 50;
									Xaxis.Update := TRUE;
									Xaxis.MoveAbsolute := TRUE;
									IF Xaxis.InPosition THEN;
										Xaxis.Update := FALSE;
										Xaxis.MoveAbsolute := FALSE;
										CncParameters_3Axis.ProgramName := 'WProg';
										MpCnc3Axis_0.Update := TRUE;
										MpCnc3Axis_0.MoveProgram := TRUE;
										IF MpCnc3Axis_0.MoveDone THEN
											MpCnc3Axis_0.Update := FALSE;
											MpCnc3Axis_0.MoveProgram := FALSE;
											X_param.Position := LengthEnd;
											Xaxis.Update := TRUE;
											Xaxis.MoveAbsolute := TRUE;
											IF Xaxis.InPosition  THEN
												Xaxis.Update := FALSE;
												Xaxis.MoveAbsolute := FALSE;
												IF StopMode THEN
													AutomaticON := FALSE;
													gdoProcessLamp := FALSE;
													NumOfElem := 0;
													WorkingMode := STOP;////////going to stop mode after completing program
												ELSE
													gdoProcessLamp := FALSE;
													Elements2Done := Elements2Done + 1;
													IF (Elements2Done = NumOfElem) AND (NumOfElem <> 0.0) THEN;
														NumOfElem := 0;
														Elements2Done := 0;
														StopMode := TRUE;
														AutomaticON := FALSE;
														WorkingMode := STOP;
													ELSE
														IF NumOfElem = 0.0 THEN;
															Elements2Done := FALSE;
															AutoModeStatus := XMOVING;
														ELSE
															AutoModeStatus := XMOVING;
														END_IF;
													END_IF;
												END_IF;

											END_IF;
										END_IF;
									END_IF;
								END_IF;
								///Program U
							ELSIF ChooseProgr = CAPITAL_U  THEN
								IF ObjLength < 115 THEN
									Elem2Small := TRUE;
									gdoProcessLamp := FALSE;
									AutoModeStatus := XMOVING;
								ELSE

									X_param.Position := CentreX + 37.5;
									Xaxis.Update := TRUE;
									Xaxis.MoveAbsolute := TRUE;
									IF Xaxis.InPosition THEN;
										Xaxis.Update := FALSE;
										Xaxis.MoveAbsolute := FALSE;
										CncParameters_3Axis.ProgramName := 'UProg';
										MpCnc3Axis_0.Update := TRUE;
										MpCnc3Axis_0.MoveProgram := TRUE;
										IF MpCnc3Axis_0.MoveDone THEN
											MpCnc3Axis_0.Update := FALSE;
											MpCnc3Axis_0.MoveProgram := FALSE;
											X_param.Position := LengthEnd;
											Xaxis.Update := TRUE;
											Xaxis.MoveAbsolute := TRUE;
											IF Xaxis.InPosition THEN
												Xaxis.Update := FALSE;
												Xaxis.MoveAbsolute := FALSE;
												IF StopMode THEN
													AutomaticON := FALSE;
													gdoProcessLamp := FALSE;
													NumOfElem := 0;
													WorkingMode := STOP;////////going to stop mode after completing program
												ELSE
													gdoProcessLamp := FALSE;
													Elements2Done := Elements2Done + 1;
													IF (Elements2Done = NumOfElem) AND (NumOfElem <> 0.0) THEN;
														NumOfElem := 0;
														Elements2Done := 0;
														StopMode := TRUE;
														AutomaticON := FALSE;
														WorkingMode := STOP;
													ELSE
														IF NumOfElem = 0.0 THEN;
															Elements2Done := FALSE;
															AutoModeStatus := XMOVING;
														ELSE
															AutoModeStatus := XMOVING;
														END_IF;
													END_IF;
												END_IF;

											END_IF;
										END_IF;
									END_IF;
								END_IF;
								//Program X
							ELSIF ChooseProgr = CAPITAL_X THEN
								IF ObjLength < 115 THEN
									Elem2Small := TRUE;
									gdoProcessLamp := FALSE;
									AutoModeStatus := XMOVING;
								ELSE

									X_param.Position := CentreX + 37.5;
									Xaxis.Update := TRUE;
									Xaxis.MoveAbsolute := TRUE;
									IF  Xaxis.InPosition THEN;
										Xaxis.Update := FALSE;
										Xaxis.MoveAbsolute := FALSE;
										CncParameters_3Axis.ProgramName := 'XProg';
										MpCnc3Axis_0.Update := TRUE;
										MpCnc3Axis_0.MoveProgram := TRUE;
										IF MpCnc3Axis_0.MoveDone THEN;
											MpCnc3Axis_0.Update := FALSE;
											MpCnc3Axis_0.MoveProgram := FALSE;
											X_param.Position := LengthEnd;
											Xaxis.Update := TRUE;
											Xaxis.MoveAbsolute := TRUE;
											IF Xaxis.InPosition THEN
												Xaxis.Update := FALSE;
												Xaxis.MoveAbsolute := FALSE;
												IF StopMode THEN
													AutomaticON := FALSE;
													gdoProcessLamp := FALSE;
													NumOfElem := 0;
													WorkingMode := STOP;////////going to stop mode after completing program
												ELSE
													gdoProcessLamp := FALSE;
													Elements2Done := Elements2Done + 1;
													IF (Elements2Done = NumOfElem) AND (NumOfElem <> 0.0) THEN;
														NumOfElem := 0;
														Elements2Done := 0;
														StopMode := TRUE;
														AutomaticON := FALSE;
														WorkingMode := STOP;
													ELSE
														IF NumOfElem = 0.0 THEN;
															Elements2Done := FALSE;
															AutoModeStatus := XMOVING;
														ELSE
															AutoModeStatus := XMOVING;
														END_IF;
													END_IF;
												END_IF;

											END_IF;
										END_IF;
									END_IF;
								END_IF;
								//Program R
							ELSIF ChooseProgr = CAPITAL_R THEN
								IF ObjLength < 90 THEN
									Elem2Small := TRUE;
									gdoProcessLamp := FALSE;
									AutoModeStatus := XMOVING;
								ELSE

									X_param.Position := CentreX + 25;
									Xaxis.Update := TRUE;
									Xaxis.MoveAbsolute := TRUE;
									IF Xaxis.InPosition THEN;
										Xaxis.Update := FALSE;
										Xaxis.MoveAbsolute := FALSE;
										CncParameters_3Axis.ProgramName := 'RProg';
										MpCnc3Axis_0.Update := TRUE;
										MpCnc3Axis_0.MoveProgram := TRUE;
										IF MpCnc3Axis_0.MoveDone THEN
											MpCnc3Axis_0.Update := FALSE;
											MpCnc3Axis_0.MoveProgram := FALSE;
											X_param.Position := LengthEnd;
											Xaxis.Update := TRUE;
											Xaxis.MoveAbsolute := TRUE;
											IF Xaxis.InPosition  THEN;
												Xaxis.Update := FALSE;
												Xaxis.MoveAbsolute := FALSE;
												IF StopMode THEN
													AutomaticON := FALSE;
													gdoProcessLamp := FALSE;
													NumOfElem := 0;
													WorkingMode := STOP;////////going to stop mode after completing program
												ELSE
													gdoProcessLamp := FALSE;
													Elements2Done := Elements2Done + 1;
													IF (Elements2Done = NumOfElem) AND (NumOfElem <> 0.0) THEN;
														NumOfElem := 0;
														Elements2Done := 0;
														StopMode := TRUE;
														AutomaticON := FALSE;
														WorkingMode := STOP;
													ELSE
														IF NumOfElem = 0.0 THEN;
															Elements2Done := FALSE;
															AutoModeStatus := XMOVING;
														ELSE
															AutoModeStatus := XMOVING;
														END_IF;
													END_IF;
												END_IF;

											END_IF;

										END_IF;
									END_IF;
								END_IF;
							END_IF;

					END_CASE

				MANUAL:
					ManualON := TRUE;
					MpCnc3Axis_0.Power := TRUE;
					IF AutomaticON THEN;
						ManualON := FALSE;
						WorkingMode := AUTOMATIC;
						JogUpX := FALSE;
						JogDownX := FALSE;
						JogUpY := FALSE;
						JogDownY := FALSE;
						JogUpZ := FALSE;
						JogUpS := FALSE;
						Saxis.JogPositive := FALSE;
					END_IF;

					IF StopMode THEN;
						ManualON := FALSE;
						WorkingMode := STOP;
						JogUpX := FALSE;
						JogDownX := FALSE;
						JogUpY := FALSE;
						JogDownY := FALSE;
						JogUpZ := FALSE;
						JogUpS := FALSE;
						Saxis.JogPositive := FALSE;

					END_IF;

					ActMode4MV := 'Manual Mode';
					IF JogModeOn THEN;
						ManualModeStatus := JOG;
					ELSE
						ManualModeStatus := PRECISE;
					END_IF;

					CASE ManualModeStatus OF
						////Chossing which axis we want to move
						PRECISE:
							IF X2Move = FALSE AND Y2Move = FALSE AND Z2Move = FALSE AND S2Move = FALSE THEN;
								Moveaxis := FALSE;
							END_IF;
							CASE AsignProp OF
								AXIS2MOVE:
									IF X2Move THEN;
											X2Move := FALSE;
											Y2Move := FALSE;
											Z2Move := FALSE;
											S2Move := FALSE;
										AsignProp := MOVEX;
									ELSIF Y2Move THEN;
											X2Move := FALSE;
											Y2Move := FALSE;
											Z2Move := FALSE;
											S2Move := FALSE;
										AsignProp := MOVEY;
									ELSIF Z2Move THEN;
											X2Move := FALSE;
											Y2Move := FALSE;
											Z2Move := FALSE;
											S2Move := FALSE;
										AsignProp := MOVEZ;
									ELSIF S2Move THEN;
											X2Move := FALSE;
											Y2Move := FALSE;
											Z2Move := FALSE;
											S2Move := FALSE;
										AsignProp := MOVES;
									END_IF;
								MOVEX:
									IF Moveaxis THEN;

										X_param.Velocity := ManXVel;
										X_param.Position := ManXPos;
										Xaxis.MoveAbsolute := TRUE;
										Moveaxis := TRUE;
										X2Move := TRUE;
										IF Xaxis.Position = ManXPos THEN;
											Moveaxis := FALSE;
											Xaxis.MoveAbsolute := FALSE;
											X2Move := FALSE;
											AsignProp := AXIS2MOVE;
										END_IF;
									END_IF;
								MOVEY:
									IF Moveaxis THEN;
										Y2Move := TRUE;
										Y_param.Velocity := ManYVel;
										Y_param.Position := ManYPos;
										Yaxis.MoveAbsolute := TRUE;
										Moveaxis := TRUE;
										IF Yaxis.Position = ManYPos THEN;
											Moveaxis := FALSE;
											Yaxis.MoveAbsolute := FALSE;
											Y2Move := FALSE;
											AsignProp := AXIS2MOVE;
										END_IF;
									END_IF;
								MOVEZ:
									IF Moveaxis THEN;
										Z2Move := TRUE;
										Z_param.Velocity := ManZVel;
										Z_param.Position := ManZPos;
										Zaxis.MoveAbsolute := TRUE;
										Moveaxis := TRUE;
										IF Zaxis.Position = ManZPos THEN;
											Moveaxis := FALSE;
											Zaxis.MoveAbsolute := FALSE;
											Z2Move := FALSE;
											AsignProp := AXIS2MOVE;
										END_IF;
									END_IF;
								MOVES:
									IF Moveaxis THEN;
										S2Move := TRUE;
										S_param.Velocity := ManSVel;
										S_param.Position := ManSPos;
										Saxis.MoveAbsolute := TRUE;
										Moveaxis := TRUE;
										IF Saxis.Position = ManSPos THEN;
											Moveaxis := FALSE;
											Saxis.MoveAbsolute := FALSE;
											S2Move := FALSE;
											AsignProp := AXIS2MOVE;
										END_IF;
									END_IF;
							END_CASE
						JOG:
							CASE JogStatus OF
								JOGTYPE:
									IF JogUpX THEN;
										JogStatus := XUP;
									ELSIF JogDownX THEN;
										JogStatus := XDOWN;
									ELSIF JogUpY THEN;
										JogStatus := YUP;
									ELSIF JogDownY THEN;
										JogStatus := YDOWN;
									ELSIF JogUpZ THEN;
										JogStatus := ZUP;
									ELSIF JogDownZ THEN;
										JogStatus := ZDOWN;
									END_IF;
								XUP:
									JogDownX := FALSE;
									JogUpY := FALSE;
									JogDownY := FALSE;
									JogUpZ := FALSE;
									JogDownZ := FALSE;
									Xaxis.JogPositive := TRUE;
									Xaxis.JogNegative := FALSE;
									Yaxis.JogPositive := FALSE;
									Yaxis.JogNegative := FALSE;
									Zaxis.JogPositive := FALSE;
									Zaxis.JogNegative := FALSE;
									IF JogUpX = FALSE THEN;
										Xaxis.JogPositive := FALSE;
										JogStatus := JOGTYPE;
									END_IF;
								XDOWN:
									JogUpX := FALSE;
									JogUpY := FALSE;
									JogDownY := FALSE;
									JogUpZ := FALSE;
									JogDownZ := FALSE;
									Xaxis.JogPositive := FALSE;
									Xaxis.JogNegative := TRUE;
									Yaxis.JogPositive := FALSE;
									Yaxis.JogNegative := FALSE;
									Zaxis.JogPositive := FALSE;
									Zaxis.JogNegative := FALSE;
									IF JogDownX = FALSE THEN;
										Xaxis.JogNegative := FALSE;
										JogStatus := JOGTYPE;
									END_IF;
								YUP:
									JogUpX := FALSE;
									JogDownX := FALSE;
									JogDownY := FALSE;
									JogUpZ := FALSE;
									JogDownZ := FALSE;
									Xaxis.JogPositive := FALSE;
									Xaxis.JogNegative := FALSE;
									Yaxis.JogPositive := TRUE;
									Yaxis.JogNegative := FALSE;
									Zaxis.JogPositive := FALSE;
									Zaxis.JogNegative := FALSE;
									IF JogUpY = FALSE THEN;
										Yaxis.JogPositive := FALSE;
										JogStatus := JOGTYPE;
									END_IF;
								YDOWN:
									JogUpX := FALSE;
									JogDownX := FALSE;
									JogUpY := FALSE;
									JogUpZ := FALSE;
									JogDownZ := FALSE;
									Xaxis.JogPositive := FALSE;
									Xaxis.JogNegative := FALSE;
									Yaxis.JogPositive := FALSE;
									Yaxis.JogNegative := TRUE;
									Zaxis.JogPositive := FALSE;
									Zaxis.JogNegative := FALSE;
									IF JogDownY = FALSE OR (Yaxis.Position = -100.0) THEN;
										Yaxis.JogNegative := FALSE;
										JogStatus := JOGTYPE;
									END_IF;
								ZUP:
									JogUpX := FALSE;
									JogDownX := FALSE;
									JogUpY := FALSE;
									JogDownY := FALSE;
									JogDownZ := FALSE;
									Xaxis.JogPositive := FALSE;
									Xaxis.JogNegative := FALSE;
									Yaxis.JogPositive := FALSE;
									Yaxis.JogNegative := FALSE;
									Zaxis.JogPositive := TRUE;
									Zaxis.JogNegative := FALSE;
									IF JogUpZ = FALSE THEN;
										Zaxis.JogPositive := FALSE;
										JogStatus := JOGTYPE;
									END_IF;
								ZDOWN:
									JogUpX := FALSE;
									JogDownX := FALSE;
									JogUpY := FALSE;
									JogDownY := FALSE;
									JogUpZ := FALSE;
									Xaxis.JogPositive := FALSE;
									Xaxis.JogNegative := FALSE;
									Yaxis.JogPositive := FALSE;
									Yaxis.JogNegative := FALSE;
									Zaxis.JogPositive := FALSE;
									Zaxis.JogNegative := TRUE;
									IF JogDownZ = FALSE THEN;
										Zaxis.JogNegative := FALSE;
										JogStatus := JOGTYPE;
									END_IF;
							END_CASE

							IF JogUpS THEN;
								Saxis.JogPositive := TRUE;
							ELSE
								Saxis.JogPositive := FALSE;
							END_IF;

					END_CASE
					///////////
					///////////////////

					//////////////////////
					////////////////////
				STOP:
					ActMode4MV := 'STOP Mode';
					Xaxis.Stop := TRUE;
					Yaxis.Stop := TRUE;
					Zaxis.Stop := TRUE;
					Saxis.Stop := TRUE;
					IF (StopMode = FALSE) AND (Xaxis.Stop = TRUE) AND (Yaxis.Stop = TRUE) AND (Zaxis.Stop = TRUE) AND (Saxis.Stop = TRUE) THEN
						IF (AutomaticON = TRUE) AND (ManualON = FALSE) THEN;
							Xaxis.Stop := FALSE;
							Yaxis.Stop := FALSE;
							Zaxis.Stop := FALSE;
							Saxis.Stop := FALSE;
							IF (Xaxis.Stop = FALSE) AND (Yaxis.Stop = FALSE) AND (Zaxis.Stop = FALSE) AND (Saxis.Stop = FALSE) THEN;
								WorkingMode := AUTOMATIC;
								AutoModeStatus := XMOVING;
							END_IF;
						ELSIF (AutomaticON = FALSE) AND (ManualON = TRUE) THEN;
							WorkingMode := MANUAL;
							Xaxis.Stop := FALSE;
							Yaxis.Stop := FALSE;
							Zaxis.Stop := FALSE;
							Saxis.Stop := FALSE;
							IF (Xaxis.Stop = FALSE) AND (Yaxis.Stop = FALSE) AND (Zaxis.Stop = FALSE) AND (Saxis.Stop = FALSE) THEN;
								WorkingMode := MANUAL;
							END_IF;
						END_IF;
					ELSIF StopMode THEN;
						AutomaticON := FALSE;
						ManualON := FALSE;

					END_IF;
					IF EDGENEG(MpCnc3Axis_0.Power) THEN;
						AutomaticON := FALSE;
						ManualON := FALSE;
						StopMode := FALSE;
						Xaxis.Update := FALSE;
						IF MpCnc3Axis_0.PowerOn = FALSE THEN;
							WorkingMode := CHOOSE_MODE;
							ServoStatus := POWER_OFF;
							Xaxis.MoveVelocity := FALSE;
						END_IF;
					END_IF;

			END_CASE

	END_CASE;
//Emergency Button
	IF EDGEPOS (EmergStop) THEN;
		MpCnc3Axis_0.Power := FALSE;
		AutomaticON := FALSE;
		ManualON := FALSE;
		StopMode := FALSE;
		Xaxis.Update := FALSE;

	END_IF
	IF  WarningSymbol1 THEN
		EmergStop := TRUE;
		MpCnc3Axis_0.Power := FALSE;
		AutomaticON := FALSE;
		ManualON := FALSE;
		StopMode := FALSE;
	END_IF;

	IF EDGENEG (WarningSymbol1) THEN
		EmergStop := FALSE;
	END_IF
	IF EDGENEG (EmergStop) THEN;
		MpCnc3Axis_0.Power := FALSE;
		WorkingMode := CHOOSE_MODE;
		ServoStatus := POWER_OFF;
		Xaxis.MoveVelocity := FALSE;
	END_IF

/////////////////////////////////////////////////

	//////////////////////////////////////
	//ALARMS
	//////////////////////////////////////
	IF EDGEPOS (EmergStop) THEN
		MpAlarmXSet (gAlarmXCore, 'EmergButton');
	END_IF
	IF EDGENEG (EmergStop) THEN
		MpAlarmXReset (gAlarmXCore, 'EmergButton');
	END_IF

	IF EDGEPOS (EmergStopAck) THEN
		MpAlarmXAcknowledge (gAlarmXCore, 'EmergButton');
		EmergStopAck := FALSE;
	END_IF

	IF EDGEPOS (Elem2Small) THEN
		MpAlarmXSet (gAlarmXCore, 'Elem2Small');
	END_IF
	IF EDGENEG (Elem2Small) THEN
		MpAlarmXReset (gAlarmXCore, 'Elem2Small');
	END_IF

	IF EDGEPOS (Elem2SmallAck) THEN
		MpAlarmXAcknowledge (gAlarmXCore, 'Elem2Small');
		Elem2SmallAck := FALSE;
	END_IF

	AckALL.Execute := AckAllButton;

	WarningSymbol1 := MpAlarmXCheckState(gAlarmXCore, 'EmergButton',mpALARMX_STATE_UNACKNOWLEDGED);
	WarningSymbol2 := MpAlarmXCheckState(gAlarmXCore, 'Elem2Small',mpALARMX_STATE_UNACKNOWLEDGED);

	IF WarningSymbol1 OR WarningSymbol2 THEN
		ShowWarning := TRUE;

	ELSE
		ShowWarning := FALSE;

	END_IF;
	///////////////////////////////////////////

	/////////////////////////////////////////
	//Milling Lamp
	//////////////////////

	IF Saxis.Velocity = 0.0 THEN;
		gdoMillingLamp := FALSE;
	ELSE
		gdoMillingLamp := TRUE;
	END_IF;

	////////////////////////////////////////

	//////PLC Open State

	//Xaxis
	IF Xaxis.Info.PLCopenState = 0 THEN;
		XState := 'mpAXIS_DISABLED';
		XOff := FALSE;
		XOn := FALSE;
		Xmove := FALSE;
	ELSIF Xaxis.Info.PLCopenState = 1 THEN;
		XState := 'mpAXIS_STANDSTILL';
		XOff := FALSE;
		XOn := TRUE;
		Xmove := FALSE;
	ELSIF Xaxis.Info.PLCopenState = 2 THEN;
		XState := 'mpAXIS_ERRORSTOP';
		XOff := FALSE;
		XOn := FALSE;
		Xmove := FALSE;
	ELSIF Xaxis.Info.PLCopenState = 3 THEN;
		XState := 'mpAXIS_STOPPING';
		XOff := TRUE;
		XOn := FALSE;
		Xmove := FALSE;
	ELSIF Xaxis.Info.PLCopenState = 4 THEN;
		XState := 'mpAXIS_DISCRETE_MOTION';
		XOff := FALSE;
		XOn := FALSE;
		Xmove := FALSE;
	ELSIF Xaxis.Info.PLCopenState = 5 THEN;
		XState := 'mpAXIS_CONTINUOUS_MOTION';
		XOff := FALSE;
		XOn := FALSE;
		Xmove := TRUE;
	ELSIF Xaxis.Info.PLCopenState = 6 THEN;
		XState := 'mpAXIS_SYNCHRONIZED_MOTION';
		XOff := FALSE;
		XOn := FALSE;
		Xmove := TRUE;
	ELSIF Xaxis.Info.PLCopenState = 7 THEN;
		XState := 'mpAXIS_HOMING';
		XOff := FALSE;
		XOn := FALSE;
		Xmove := FALSE;
	END_IF;

	//Yaxis
	IF Yaxis.Info.PLCopenState = 0 THEN;
		YState := 'mpAXIS_DISABLED';
		YOff := FALSE;
		YOn := FALSE;
		Ymove := FALSE;
	ELSIF Yaxis.Info.PLCopenState = 1THEN;
		YState := 'mpAXIS_STANDSTILL';
		YOff := FALSE;
		YOn := TRUE;
		Ymove := FALSE;
	ELSIF Yaxis.Info.PLCopenState = 2 THEN;
		YState := 'mpAXIS_ERRORSTOP';
		YOff := FALSE;
		YOn := FALSE;
		Ymove := FALSE;
	ELSIF Yaxis.Info.PLCopenState = 3 THEN;
		YState := 'mpAXIS_STOPPING';
		YOff := TRUE;
		YOn := FALSE;
		Ymove := FALSE;
	ELSIF Yaxis.Info.PLCopenState = 4 THEN;
		YState := 'mpAXIS_DISCRETE_MOTION';
		YOff := FALSE;
		YOn := FALSE;
		Ymove := FALSE;
	ELSIF Yaxis.Info.PLCopenState = 5 THEN;
		YState := 'mpAXIS_CONTINUOUS_MOTION';
		YOff := FALSE;
		YOn := FALSE;
		Ymove := TRUE;
	ELSIF Xaxis.Info.PLCopenState = 6 THEN;
		YState := 'mpAXIS_SYNCHRONIZED_MOTION';
		YOff := FALSE;
		YOn := FALSE;
		Ymove := TRUE;
	ELSIF Xaxis.Info.PLCopenState = 7 THEN;
		YState := 'mpAXIS_HOMING';
		YOff := FALSE;
		YOn := FALSE;
		Ymove := FALSE;
	END_IF;

	//Zaxis
	IF Zaxis.Info.PLCopenState = 0 THEN;
		ZState := 'mpAXIS_DISABLED';
		ZOff := FALSE;
		ZOn := FALSE;
		Zmove := FALSE;
	ELSIF Zaxis.Info.PLCopenState = 1 THEN;
		ZState := 'mpAXIS_STANDSTILL';
		ZOff := FALSE;
		ZOn := TRUE;
		Zmove := FALSE;
	ELSIF Zaxis.Info.PLCopenState = 2 THEN;
		ZState := 'mpAXIS_ERRORSTOP';
		ZOff := FALSE;
		ZOn := FALSE;
		Zmove := FALSE;
	ELSIF Zaxis.Info.PLCopenState = 3 THEN;
		ZState := 'mpAXIS_STOPPING';
		ZOff := TRUE;
		ZOn := FALSE;
		Zmove := FALSE;
	ELSIF Zaxis.Info.PLCopenState = 4 THEN;
		ZState := 'mpAXIS_DISCRETE_MOTION';
		ZOff := FALSE;
		ZOn := FALSE;
		Zmove := FALSE;
	ELSIF Zaxis.Info.PLCopenState = 5 THEN;
		ZState := 'mpAXIS_CONTINUOUS_MOTION';
		ZOff := FALSE;
		ZOn := FALSE;
		Zmove := TRUE;
	ELSIF Zaxis.Info.PLCopenState = 6 THEN;
		ZState := 'mpAXIS_SYNCHRONIZED_MOTION';
		ZOff := FALSE;
		ZOn := FALSE;
		Zmove := TRUE;
	ELSIF Zaxis.Info.PLCopenState = 7 THEN;
		ZState := 'mpAXIS_HOMING';
		ZOff := FALSE;
		ZOn := FALSE;
		Zmove := FALSE;
	END_IF;

	//Saxis
	IF Saxis.Info.PLCopenState = 0 THEN;
		SState := 'mpAXIS_DISABLED';
		SOff := FALSE;
		SOn := FALSE;
		Smove := FALSE;
	ELSIF Saxis.Info.PLCopenState = 1 THEN;
		SState := 'mpAXIS_STANDSTILL';
		SOff := FALSE;
		SOn := TRUE;
		Smove := FALSE;
	ELSIF Saxis.Info.PLCopenState = 2 THEN;
		SState := 'mpAXIS_ERRORSTOP';
		SOff := FALSE;
		SOn := FALSE;
		Smove := FALSE;
	ELSIF Saxis.Info.PLCopenState = 3 THEN;
		SState := 'mpAXIS_STOPPING';
		SOff := TRUE;
		SOn := FALSE;
		Smove := FALSE;
	ELSIF Saxis.Info.PLCopenState = 4 THEN;
		SState := 'mpAXIS_DISCRETE_MOTION';
		SOff := FALSE;
		SOn := FALSE;
		Smove := FALSE;
	ELSIF Saxis.Info.PLCopenState = 5 THEN;
		SState := 'mpAXIS_CONTINUOUS_MOTION';
		SOff := FALSE;
		SOn := FALSE;
		Smove := TRUE;
	ELSIF Saxis.Info.PLCopenState = 6 THEN;
		SState := 'mpAXIS_SYNCHRONIZED_MOTION';
		SOff := FALSE;
		SOn := FALSE;
		Smove := TRUE;
	ELSIF Saxis.Info.PLCopenState = 7 THEN;
		SState := 'mpAXIS_HOMING';
		SOff := FALSE;
		SOn := FALSE;
		Smove := FALSE;
	END_IF;

	//////////////////////////////////////////////////////////////////////
	//////////////////////////////////////////////////////////////////////
	MpCnc3Axis_0();
	Xaxis();
	Yaxis();
	Zaxis();
	Saxis();
	MpAlarmXCore_0();
	AckALL();
	MpAlarmXHistory_0();

END_PROGRAM

PROGRAM _EXIT

	//Alarms
	MpAlarmXCore_0.Enable := FALSE;
	MpAlarmXCore_0();

	AckALL.Enable := FALSE;
	AckALL();

	MpAlarmXHistory_0.Enable := FALSE;
	MpAlarmXHistory_0();

	//3 Axis
	MpCnc3Axis_0.Power  := FALSE;
	MpCnc3Axis_0.Home   := FALSE;
	MpCnc3Axis_0.Enable := FALSE;
	MpCnc3Axis_0();
	/////

	//X axis
	Xaxis.Power  := FALSE;
	Xaxis.Home   := FALSE;
	Xaxis.MoveAbsolute := FALSE;
	Xaxis.MoveAdditive := FALSE;
	Xaxis.MoveVelocity := FALSE;
	Xaxis.Stop         := FALSE;
	Xaxis.ErrorReset   := FALSE;
	Xaxis();
	Xaxis.Enable := FALSE;
	Xaxis();
	/////////////////

	//Y axis
	Xaxis.Power  := FALSE;
	Xaxis.Home   := FALSE;
	Xaxis.MoveAbsolute := FALSE;
	Xaxis.MoveAdditive := FALSE;
	Xaxis.MoveVelocity := FALSE;
	Xaxis.Stop         := FALSE;
	Xaxis.ErrorReset   := FALSE;
	Xaxis();
	Xaxis.Enable := FALSE;
	Xaxis();
	/////////////////

	//Z axis
	Xaxis.Power  := FALSE;
	Xaxis.Home   := FALSE;
	Xaxis.MoveAbsolute := FALSE;
	Xaxis.MoveAdditive := FALSE;
	Xaxis.MoveVelocity := FALSE;
	Xaxis.Stop         := FALSE;
	Xaxis.ErrorReset   := FALSE;
	Xaxis();
	Xaxis.Enable := FALSE;
	Xaxis();
	/////////////////

	//S axis
	Xaxis.Power  := FALSE;
	Xaxis.Home   := FALSE;
	Xaxis.MoveAbsolute := FALSE;
	Xaxis.MoveAdditive := FALSE;
	Xaxis.MoveVelocity := FALSE;
	Xaxis.Stop         := FALSE;
	Xaxis.ErrorReset   := FALSE;
	Xaxis();
	Xaxis.Enable := FALSE;
	Xaxis();
	/////////////////

END_PROGRAM
```

### Data object Logical/CNC/IProg (Cnc)

#### IProg.cnc - CNC program (G-Code)
```
%001 (CncProgram)

N05 G90     (absolute coordinates)
N15 G01 Y150 F1500
N20	S10000
N25 M3
N30 G01 Z99 F1500
N35 G01 Y250 F1500
N40 M5
N45 G01 Z300 F1500
N50 G01 Y0 F1500
N999 M30
```

### Data object Logical/CNC/WProg (Cnc)

#### WProg.cnc - CNC program (G-Code)
```
%001 (CncProgram)

N05 G91     (absolute coordinates)
N15 G01 Y250 F1500
N20	S10000
N25 M3
N30 G01 Z-201 F1500
N35 G01 X25 Y-100 F1500
N40 G01 X25 Y50 F1500
N45 G01 X25 Y-50 F1500
N50 G01 X25 Y100 F1500
N65 M5
N70 G01 Z201 F1500
N75 G01 X100 Y-250 F1500
N999 M30
```

### Data object Logical/CNC/UProg (Cnc)

#### UProg.cnc - CNC program (G-Code)
```
%001 (CncProgram)

N05 G91
N10 G17   (absolute coordinates)
N15 G01 Y250 F1500
N20	S10000
N25 M3
N30 G01 Z-201 F1500
N35 G01 Y-75 F1500
N40 G02 X-25 Y-25 I-25 F1500
N45 G01 X-25 F500
N50 G02 X-25  Y25  J25 F1500
N55 G01 Y75	 F1500
N65 M5
N70 G01 Z201 F1500
N75 G01 X75 Y-250 F1500
N999 M30
```

### Data object Logical/CNC/isProg (Cnc)

#### isProg.cnc - CNC program (G-Code)
```
%001 (CncProgram)

N05 G90     (absolute coordinates)
(N10 G21)    	(programming in milimeters mm)
N15 G01 Y150 F1500
N20	S10000
N25 M3
N30 G01 Z99 F1500
N35 G01 Y225 F1500
N40 M5
N45 G01 Z300 F1500
N50 G01 Y250 F1500
N55	S10000
N60 M3
N65 G01 Z99 F1500
N70 M5
N75 G01 Z300 F1500
N80 G01 Y0 F1500
N999 M30
```

### Data object Logical/CNC/XProg (Cnc)

#### XProg.cnc - CNC program (G-Code)
```
%001 (CncProgram)

N05 G91     (absolute coordinates)
N15 G01 Y250 F1500
N20	S10000
N25 M3
N30 G01 Z-201 F1500
N35 G01 X-75 Y-100 F1500
N40 M5
N45 G01 Z201 F1500
N50 G01 Y100 F1500
N65	S10000
N70 M3
N75 G01 Z-201 F1500
N80 G01 X75  Y-100 F1500
N85 M5
N90 G01 Z201 F1500
N95 G01 Y-150 F1500
N999 M30
```

### Data object Logical/CNC/RProg (Cnc)

#### RProg.cnc - CNC program (G-Code)
```
%001 (CncProgram)

N05 G91     (absolute coordinates)
N10 G17
N15 G01 Y150 F1500
N20	S10000
N25 M3
N30 G01 Z-201 F1500
N35 G01 Y100 F1500
N40 G01 X-25 F1500
N45 G03 Y-50 J-25 F1500
N50 G01 X25 F500
N55 G01 X-50 Y-50 F1500
N65 M5
N70 G01 Z201 F1500
N75 G01 Y-150 F1500
N999 M30
```

- Visualisation Logical/mappView (not shown)

- Project.language (not shown)

Listed in the project but not available here: Logical/Source
